DEVICE_TYPE _TCREST
  (* Standard: 61499-2 *)
  (* Version 0.1, 2017-00-09, hpea485, UOA *)
  RESOURCE c0 : _Core0
  END_RESOURCE
  RESOURCE c1 : _Core1
  END_RESOURCE
  RESOURCE c2 : _Core2
  END_RESOURCE
  RESOURCE c3 : _Core3
  END_RESOURCE
END_DEVICE_TYPE
